PROGRAM POU_MULTPLY
VAR
	Result:REAL;
	Value01:REAL;
	Value02:REAL;
END_VAR

Result:=MAIN.Value01*MAIN.Value02;

END_PROGRAM

(* stored: Version 1.1.0.1, ProductVersion 3.1.4024.4
   POU POU_MULTPLY: Id {7e870540-0b56-4953-b691-6ecc0b2c616f}, SpecialFunc None *)
